// TIA Portal V19 export
DATA_BLOCK "hmiDatatransferTP1200"   // DB10
{ S7_Optimized_Access := 'TRUE' }
// stored: AutoNumber false, MemoryReserve 100
   VAR
      plc1LedState : Int;
      plc2LedState : Int;
      plcOperationState : Int;
      plcMrpState : Int;
      plcStopMonitoring : Int;
   END_VAR
BEGIN
END_DATA_BLOCK
